TYPE ST_InputStationHSControlOP11601 :
STRUCT
	{attribute 'OPC.UA.DA.Description' := 'Dummy (for making struct visible on OPC UA'}
	Dummy						: BOOL;
END_STRUCT
END_TYPE

(* stored: Version 1.1.0.1, ProductVersion 3.1.4024.2
   DUT ST_InputStationHSControlOP11601: Id {495bb13b-8384-4aba-84af-a1b40bda9a22} *)
